// TIA Portal V18 export
DATA_BLOCK "ROBOT_COMMUNICATION_DB"   // DB2
{ S7_Optimized_Access := 'FALSE' }
   VAR
      adapters : Array[0..0] of "LCCF_typeEnetAdaptConfig_1";
      datas { S7_SetPoint := 'True'} : Array[0..0] of "LCCF_typeEnetAdaptData_1";
      connection_OK { S7_SetPoint := 'True'} : Bool;
      connection_ERROR : Bool;
   END_VAR
BEGIN
   adapters[0].address.ADDR[1] := 192;
   adapters[0].address.ADDR[2] := 168;
   adapters[0].address.ADDR[3] := 0;
   adapters[0].address.ADDR[4] := 10;
   adapters[0].vendorIdentifier := 356;
   adapters[0].productType := 12;
   adapters[0].productCode := 2;
   adapters[0].revisionMajor := 2;
   adapters[0].revisionMinor := 2;
   adapters[0].assemblyInstance := 100;
   adapters[0].packetInterval := T#32ms;
   adapters[0].conPointOutputIdentifier := 153;
   adapters[0].conPointOutputSize := 16;
   adapters[0].conPointInputIdentifier := 103;
   adapters[0].conPointInputSize := 16;
END_DATA_BLOCK
